FUNCTION_BLOCK OneTestHasMissingTest EXTENDS FB_TestSuite

METHOD TestNameIsDifferent
IF TEST_ORDERED('WithTimestampZeroTimeExpectCurrentTime') THEN
    fbFunctionBlockUnderTest(Parameters);
 
    AssertEquals(Expected := 'SomeValue',
                 Actual := fbFunctionBlockUnderTest.OutVariable,
                 Message := 'Test failed');
 
    TEST_FINISHED();
END_IF
END_METHOD

END_FUNCTION_BLOCK

(* stored: Version 1.1.0.1, ProductVersion 3.1.4024.12
   POU OrderedTest: Id {730f5b54-1f58-0e36-3ed6-13b8b66d32c3}, SpecialFunc None
   Method TestNameIsDifferent: Id {e7546a67-4e1f-0a30-2978-e2d2f1e39ace} *)
